FUNCTION_BLOCK FB_StateMachine
VAR_INPUT
END_VAR
VAR_OUTPUT
END_VAR
VAR
	eState : E_State;
	xManualEnable : BOOL;
	xUnitEnable : BOOL;
	xCoilClean : BOOL;
	xEmergencyFlag : BOOL;
	xCoilCleanFinished : BOOL;
	xFirstCycle: BOOL := TRUE;
END_VAR

IF xFirstCycle THEN 
	eState := E_State.Off;
END_IF
	


CASE eState OF
	
	E_State.Off :
		IF xManualEnable THEN eState := E_State.Manual;
		ELSIF xUnitEnable THEN eState := E_State.Auto;
		END_IF
	
	E_State.Auto :
	 	IF xEmergencyFlag THEN eState := E_State.Emergency;
		ELSIF xManualEnable THEN eState := E_State.Manual;
		ELSIF NOT xUnitEnable THEN eState := E_State.Off;
		END_IF 
	
	E_State.Manual :
		IF NOT xManualEnable THEN eState := E_State.Off;
		ELSIF xCoilClean THEN eState := E_State.CoilClean;					
		END_IF
	
	E_State.CoilClean :
		IF xEmergencyFlag THEN eState := E_State.Emergency;
		ELSIF xCoilCleanFinished THEN eState := E_State.Manual;
									  xCoilClean := FALSE;
									  xCoilCleanFinished := FALSE;								
		END_IF
	
	E_State.Emergency :
		IF NOT xEmergencyFlag THEN eState := E_State.Off;
		END_IF

END_CASE

xFirstCycle := FALSE;

END_FUNCTION_BLOCK

(* stored: Version 1.1.0.1, ProductVersion 3.1.4024.11
   POU FB_StateMachine: Id {8b9038d6-4ca9-4706-96f5-cc1139cf3fcb}, SpecialFunc None *)
